// TIA Portal project "Fase4_Rodrigo_lorenzo" (V17)

(* hardware
DEVICE "S7-1200 station_1"  S7-1200 Station
   slot 0: "Rack_0"  S7-1200 Rack  Rack  V1.0
   slot 1: "PLC_1"  CPU 1214C AC/DC/Rly  6ES7 214-1BE30-0XB0  V2.2
*)

// ===== PLC "PLC_1"  CPU 1214C AC/DC/Rly =====

VAR_GLOBAL   // PLC tag table "Default tag table"
   "+" AT %M100.0 : Bool;
   "-" AT %M100.1 : Bool;
   "Semaforo_Rojo" AT %Q0.1 : Bool;
   "Contador" AT %MW100 : Int;
   "Semaforo_Amarillo" AT %Q0.3 : Bool;
   "Semaforo_Verde" AT %Q0.6 : Bool;
END_VAR

// folder: System blocks/Program resources

DATA_BLOCK "Contador_Coches"   // DB2
{ S7_Optimized_Access := 'TRUE' }
AUTHOR : Simatic
FAMILY : IEC
NAME : CNTR
VERSION : 1.0
// stored: InstanceOfName IEC_COUNTER
"IEC_COUNTER"
BEGIN
END_DATA_BLOCK

// folder: (top level)

ORGANIZATION_BLOCK "Main"   // OB1, LAD, ProgramCycle
TITLE = "Main Program Sweep (Cycle)"
{ S7_Optimized_Access := 'TRUE' }
VERSION : 0.1
BEGIN

REGION Network 1
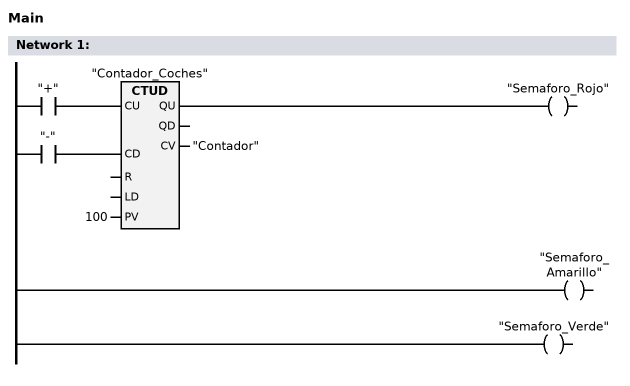
   "Contador_Coches".CTUD(CU := "+", CD := "-", PV := 100, CV => "Contador");
   "Semaforo_Rojo" := "Contador_Coches".QU;
   "Semaforo_Amarillo" := TRUE;
   "Semaforo_Verde" := TRUE;
END_REGION
END_ORGANIZATION_BLOCK